// TIA Portal V20 export
TYPE "LER_typeResetReaderUDT"
// stored: Access Published
   STRUCT
      Input : Struct
         execute : Bool;
      END_STRUCT;
      Output : Struct
         done : Bool;
         busy : Bool;
         error : Bool;
         status : DWord;
      END_STRUCT;
   END_STRUCT;
END_TYPE
